(*
SPDX-FileCopyrightText: © 2026 Oleksandr Tiutyk <trofimich@gmail.com>
SPDX-License-Identifier: MIT
License: https://opensource.org/license/mit
*)

(*!
<summary>Defines the operational lifecycle states of an automation component.</summary>
*)

{attribute 'qualified_only'}
{attribute 'strict'}
{attribute 'to_string'}
TYPE OPERATIONAL_STATE :
(
	INITIALIZING := 0, (*!<description>Start state for self and children initialization.</description>*)
	WORKING,           (*!<description>Normal working mode after successful initialization.</description>*)
	(*!
	<description>
	Recoverable stopped state. Entered after Stop or critical runtime error. Reset required to return to WORKING.
	</description>
	*)
	STOPPED,
	INVALID            (*!<description>Any error occurred during initialization, final state.</description>*)
);
END_TYPE

(* stored: Version 1.1.0.1
   DUT OPERATIONAL_STATE: Id {3a7a0191-f562-4dbc-a295-c4fdddac5490} *)
